FUNCTION TryConvert_SINT_TO_DINT : BOOL
VAR_INPUT
	in : SINT;
	out : REFERENCE TO DINT;
END_VAR

out := SINT_TO_DINT(in);
TryConvert_SINT_TO_DINT := TRUE;

END_FUNCTION

(* stored: Version 1.1.0.1, ProductVersion 3.1.4024.12
   POU TryConvert_SINT_TO_DINT: Id {1b51c2eb-dbee-4f69-95aa-42d0dae10a9e}, SpecialFunc None *)
